// Mitsubishi GX Works2 project: 2023-05-25 #1 생산자동화기능사 7번   PLC: Q03UDV
// 생산자동화기능사

// global labels: Global1
VAR_GLOBAL
  PB1 AT X0 : BOOL;
  PB2 AT X1 : BOOL;
  정지 AT X2 : BOOL;
  공급후진 AT X3 : BOOL;
  공급전진 AT X4 : BOOL;
  가공후진 AT X5 : BOOL;
  가공전진 AT X6 : BOOL;
  송출후진 AT X7 : BOOL;
  송출전진 AT X8 : BOOL;
  배출후진 AT X9 : BOOL;
  배출전진 AT X0A : BOOL;
  매거진 AT X0B : BOOL;
  금속센서 AT X0F : BOOL;
  PB3 AT X0C : BOOL;
  적색 AT Y20 : BOOL;
  황색 AT Y21 : BOOL;
  녹색 AT Y22 : BOOL;
  공급1 AT Y23 : BOOL;
  공급2 AT Y24 : BOOL;
  가공 AT Y25 : BOOL;
  드릴 AT Y26 : BOOL;
  송출 AT Y27 : BOOL;
  배출 AT Y28 : BOOL;
  컨베이어 AT Y29 : BOOL;
END_VAR

PROGRAM 테스트동작
VAR
  STATE : INT;
END_VAR
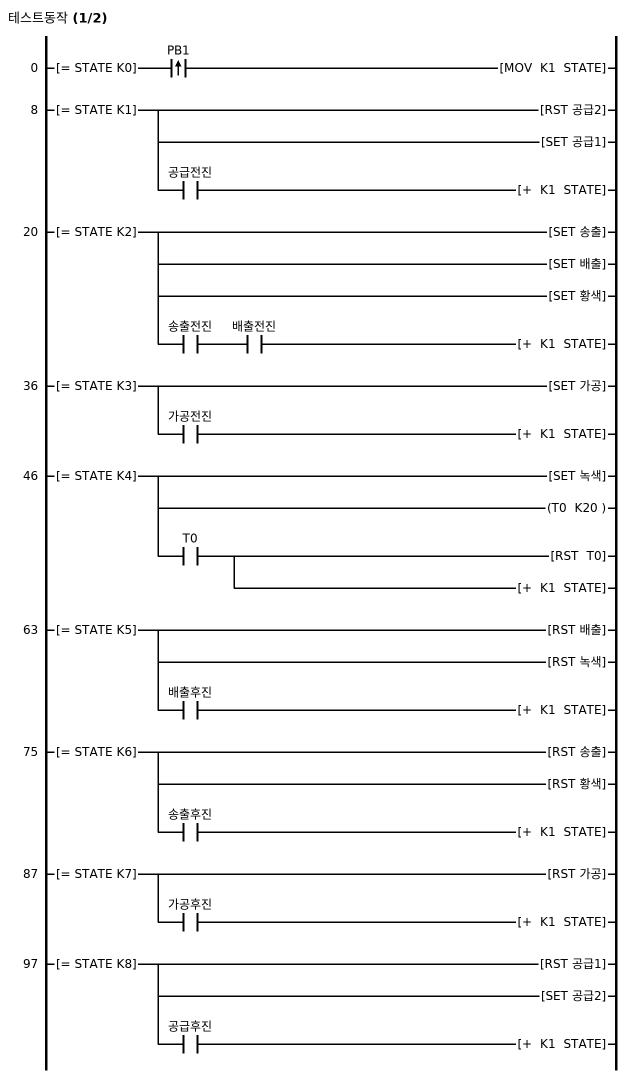
0     LD=     STATE K0
      ANDP    PB1
      MOV     K1 STATE
8     LD=     STATE K1
      RST     공급2
      SET     공급1
      AND     공급전진
      +       K1 STATE
20    LD=     STATE K2
      SET     송출
      SET     배출
      SET     황색
      AND     송출전진
      AND     배출전진
      +       K1 STATE
36    LD=     STATE K3
      SET     가공
      AND     가공전진
      +       K1 STATE
46    LD=     STATE K4
      SET     녹색
      OUT     T0 K20
      AND     T0
      RST     T0
      +       K1 STATE
63    LD=     STATE K5
      RST     배출
      RST     녹색
      AND     배출후진
      +       K1 STATE
75    LD=     STATE K6
      RST     송출
      RST     황색
      AND     송출후진
      +       K1 STATE
87    LD=     STATE K7
      RST     가공
      AND     가공후진
      +       K1 STATE
97    LD=     STATE K8
      RST     공급1
      SET     공급2
      AND     공급후진
      +       K1 STATE
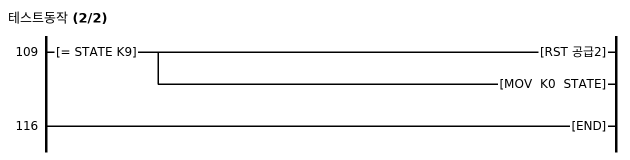
109   LD=     STATE K9
      RST     공급2
      MOV     K0 STATE
116   END
END_PROGRAM

PROGRAM 단속연속동작
VAR
  STATE : INT;
  METAL : INT;
END_VAR
VAR CONSTANT
  금속 : INT := 1;
  비금속 : INT := 2;
END_VAR
VAR
  MODE : INT;
END_VAR
VAR CONSTANT
  단속 : INT;
  연속 : INT := 1;
END_VAR
VAR
  CNT_METAL : INT;
  점멸1 : ARRAY [0..3] OF BOOL;
  STATE_EMR : INT;
  점멸2 : ARRAY [0..3] OF BOOL;
END_VAR
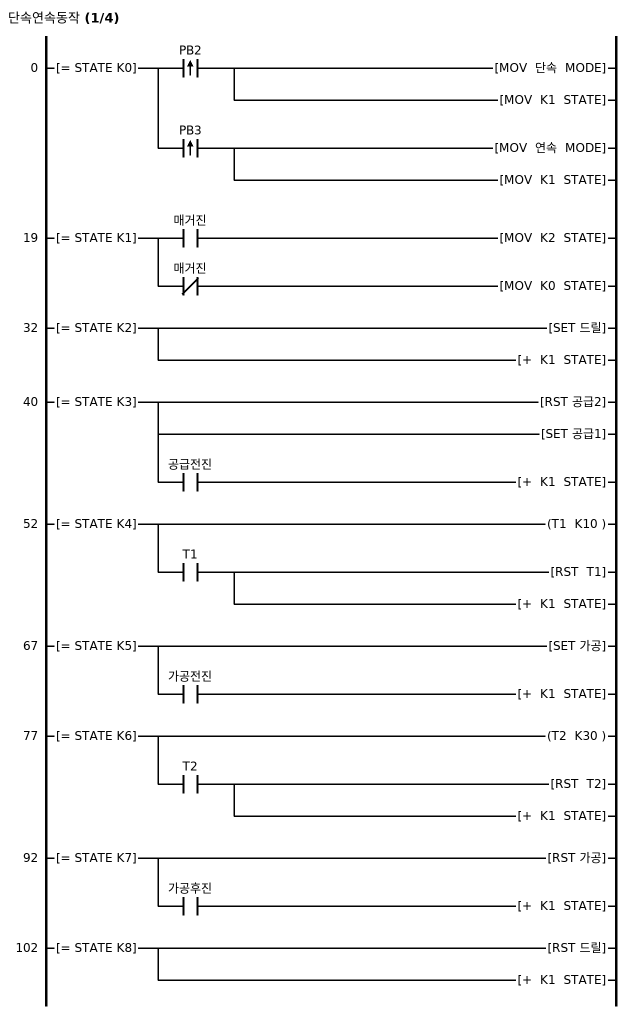
0     LD=     STATE K0
      MPS
      ANDP    PB2
      MOV     단속 MODE
      MOV     K1 STATE
      MPP
      ANDP    PB3
      MOV     연속 MODE
      MOV     K1 STATE
19    LD=     STATE K1
      MPS
      AND     매거진
      MOV     K2 STATE
      MPP
      ANI     매거진
      MOV     K0 STATE
32    LD=     STATE K2
      SET     드릴
      +       K1 STATE
40    LD=     STATE K3
      RST     공급2
      SET     공급1
      AND     공급전진
      +       K1 STATE
52    LD=     STATE K4
      OUT     T1 K10
      AND     T1
      RST     T1
      +       K1 STATE
67    LD=     STATE K5
      SET     가공
      AND     가공전진
      +       K1 STATE
77    LD=     STATE K6
      OUT     T2 K30
      AND     T2
      RST     T2
      +       K1 STATE
92    LD=     STATE K7
      RST     가공
      AND     가공후진
      +       K1 STATE
102   LD=     STATE K8
      RST     드릴
      +       K1 STATE
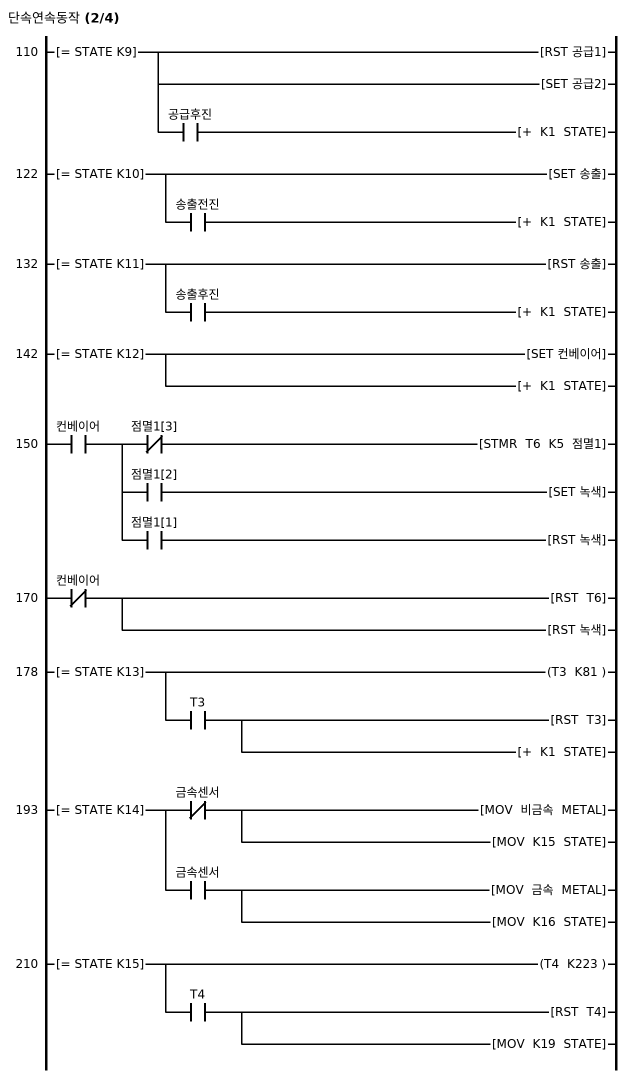
110   LD=     STATE K9
      RST     공급1
      SET     공급2
      AND     공급후진
      +       K1 STATE
122   LD=     STATE K10
      SET     송출
      AND     송출전진
      +       K1 STATE
132   LD=     STATE K11
      RST     송출
      AND     송출후진
      +       K1 STATE
142   LD=     STATE K12
      SET     컨베이어
      +       K1 STATE
150   LD      컨베이어
      MPS
      ANI     점멸1[3]
      STMR    T6 K5 점멸1
      MRD
      AND     점멸1[2]
      SET     녹색
      MPP
      AND     점멸1[1]
      RST     녹색
170   LDI     컨베이어
      RST     T6
      RST     녹색
178   LD=     STATE K13
      OUT     T3 K81
      AND     T3
      RST     T3
      +       K1 STATE
193   LD=     STATE K14
      MPS
      ANI     금속센서
      MOV     비금속 METAL
      MOV     K15 STATE
      MPP
      AND     금속센서
      MOV     금속 METAL
      MOV     K16 STATE
210   LD=     STATE K15
      OUT     T4 K223
      AND     T4
      RST     T4
      MOV     K19 STATE
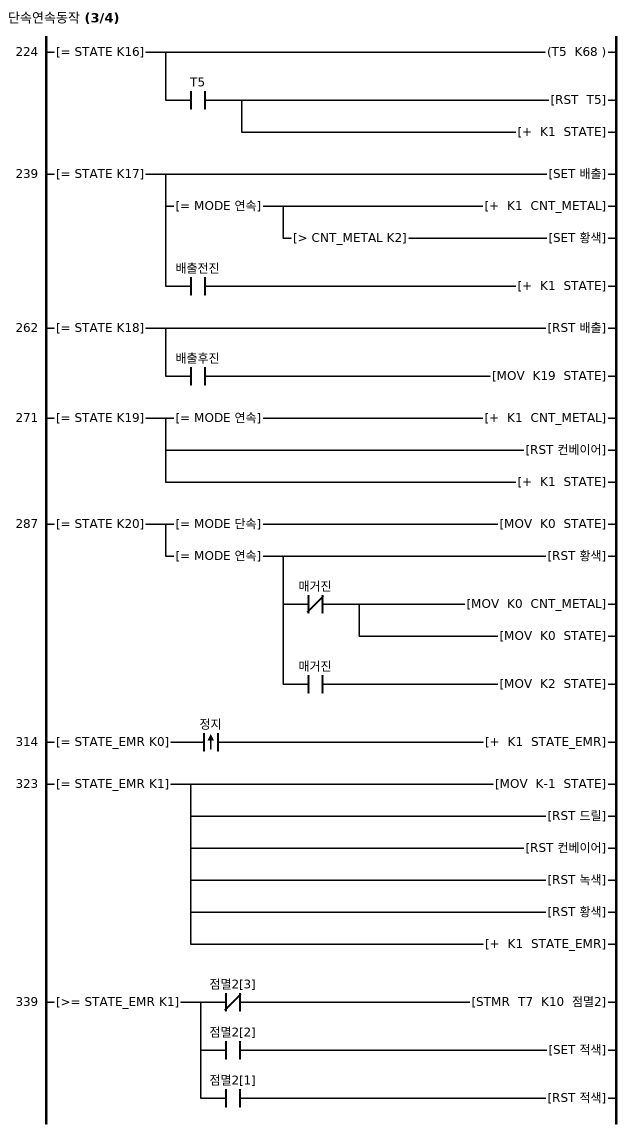
224   LD=     STATE K16
      OUT     T5 K68
      AND     T5
      RST     T5
      +       K1 STATE
239   LD=     STATE K17
      SET     배출
      MPS
      AND=    MODE 연속
      +       K1 CNT_METAL
      AND>    CNT_METAL K2
      SET     황색
      MPP
      AND     배출전진
      +       K1 STATE
262   LD=     STATE K18
      RST     배출
      AND     배출후진
      MOV     K19 STATE
271   LD=     STATE K19
      MPS
      AND=    MODE 연속
      +       K1 CNT_METAL
      MPP
      RST     컨베이어
      +       K1 STATE
287   LD=     STATE K20
      MPS
      AND=    MODE 단속
      MOV     K0 STATE
      MPP
      AND=    MODE 연속
      RST     황색
      MPS
      ANI     매거진
      MOV     K0 CNT_METAL
      MOV     K0 STATE
      MPP
      AND     매거진
      MOV     K2 STATE
314   LD=     STATE_EMR K0
      ANDP    정지
      +       K1 STATE_EMR
323   LD=     STATE_EMR K1
      MOV     K-1 STATE
      RST     드릴
      RST     컨베이어
      RST     녹색
      RST     황색
      +       K1 STATE_EMR
339   LD>=    STATE_EMR K1
      MPS
      ANI     점멸2[3]
      STMR    T7 K10 점멸2
      MRD
      AND     점멸2[2]
      SET     적색
      MPP
      AND     점멸2[1]
      RST     적색
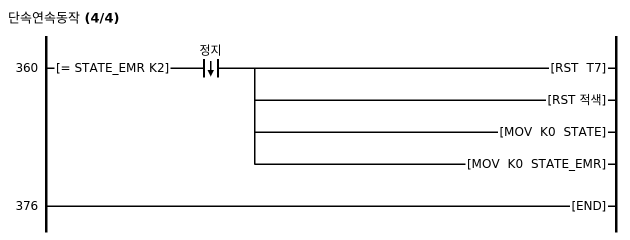
360   LD=     STATE_EMR K2
      ANDF    정지
      RST     T7
      RST     적색
      MOV     K0 STATE
      MOV     K0 STATE_EMR
376   END
END_PROGRAM
